# EPICS substitutions: iocs/MC02/db/SAI_MotorRecord.substitutions
file /opt/epics/modules/SAI/db/SAI_MotorRecord.template {
pattern {ASYNPORT,      PMACPORT,       TMOT,   PMAC_MTR,       P,              R,                      AXIS,           DESC,             MRES,       PREC,   EGU,    VEL,    TACC,      OFFS,           HSLM,           LSLM,      ALIAS}
        { "pmac",       "PMAC",         1.0,    1,              "XF:06BMA-OP",  "{Mono:DCM1-Ax:",       "Bragg}Mtr",    "Bragg",          0.000005,   6,      "deg",  0.5,    0.1,       16.05442,       42.957195,      -21.39561, dcm_bragg}
        { "pmac",       "PMAC",         1.0,    2,              "XF:06BMA-OP",  "{Mono:DCM1-Ax:",       "Bragg2}Mtr",   "Bragg Sec Enc",  0.000005,   6,      "deg",  0.5,    0.1,       16.05442,       0,              0,         dcm_bragg2}
        { "pmac",       "PMAC",         1.0,    3,              "XF:06BMA-OP",  "{Mono:DCM1-Ax:",       "P2}Mtr",       "2nd Xtal Pitch", 0.00043,    4,      "mrad", 0.42,   0.1,       6.1362,         14.1351,        -26.4075,  dcm_pitch}
        { "pmac",       "PMAC",         1.0,    4,              "XF:06BMA-OP",  "{Mono:DCM1-Ax:",       "R2}Mtr",       "2nd Xtal Roll",  0.00042,    4,      "mrad", 0.42,   0.1,       9.94056,        11.9532,        -31.8339,  dcm_roll}
        { "pmac",       "PMAC",         1.0,    5,              "XF:06BMA-OP",  "{Mono:DCM1-Ax:",       "Per2}Mtr",     "2nd Xtal Perp",  0.0001,     4,      "mm",   0.625,  0.1,       25.2427,        26.5,           1.39,      dcm_perp}
        { "pmac",       "PMAC",         1.0,    6,              "XF:06BMA-OP",  "{Mono:DCM1-Ax:",       "Par2}Mtr",     "2nd Xtal Para",  0.0001,     4,      "mm",   0.625,  0.1,       72.8658,        158.5,          12.3,      dcm_para}
        { "pmac",       "PMAC",         1.0,    7,              "XF:06BMA-OP",  "{Mono:DCM1-Ax:",       "X}Mtr",        "Goni Lateral",   0.0001,     4,      "mm",   0.5,    0.1,       0,              35.826115,      -36,       dcm_x}
        { "pmac",       "PMAC",         1.0,    8,              "XF:06BMA-OP",  "{Mono:DCM1-Ax:",       "Y}Mtr",        "Vertical",       0.0001,     5,      "mm",   0.2,    0.015625,  0,              5.0,            -5.0,      dcm_y}
#        { "pmac",       "PMAC",         1.0,    8,              "XF:06BMA-OP",  "{Mono:DCM1-Ax:",       "Y}Mtr",        "Vertical",       0.0001,     5,      "mm",   0.2,    0.015625,  0,              30.892195,      -27.18482, dcm_y}
}

## BR, 28 Nov 2017
## changed per2 offset from 20.6627 to 25.2427
## changed par2 offset from 66.3658 to 68.8658
## changed par2 HLM_SP from 155.66 to 158.5
